{attribute 'linkalways'} 
{attribute 'no_explicit_call' := 'This FB is a CLASS and must be accessed using methods or properties'}
{attribute 'enable_dynamic_creation'}
FUNCTION_BLOCK Node_ContainerType_Vector_TcVnRectangle_DINT EXTENDS Node
VAR
    out : _GUID;
END_VAR

METHOD PUBLIC  Clone : I_Node
VAR
	pNode : POINTER TO Node_ContainerType_Vector_TcVnRectangle_DINT;
END_VAR
pNode := __NEW(Node_ContainerType_Vector_TcVnRectangle_DINT);
Clone := pNode^;
END_METHOD

METHOD FB_init : BOOL
VAR_INPUT
	bInitRetains : BOOL; // if TRUE, the retain variables are initialized (warm start / cold start)
	bInCopyCode : BOOL;  // if TRUE, the instance afterwards gets moved into the copy code (online change)
END_VAR
AddOutput('out', out);
END_METHOD

METHOD PROTECTED OnExecute
out.Value := ContainerType_Vector_TcVnRectangle_DINT;
END_METHOD

END_FUNCTION_BLOCK

(* stored: Version 1.1.0.1, ProductVersion 3.1.4026.17
   POU Node_ContainerType_Vector_TcVnRectangle_DINT: Id {f3deff4c-9160-0cba-0fda-e10b739636b0}, SpecialFunc None
   Folder Constructor: Id {7285d3c2-6d73-0782-1e39-5fa496b23873}
   Method Clone: Id {77c6d10c-bb60-00d2-0599-d293b5ebb2fe}
   Method FB_init: Id {4ae17c91-7211-0159-1a08-abbcdfe611c9}
   Method OnExecute: Id {e276bbbe-aa74-0e61-2533-c193f27a3d03} *)
